FUNCTION "GLUE_SCALE" : VOID
TITLE =Glue Scale: DP Read, ASCII Parse, Valve Control, Alarms
// v0.11 - Simplified "Parse integer part" network: replaced the 7
//   duplicated digit-check blocks (Byte_0..Byte_6, one hand-unrolled
//   per byte, ~140 lines) with a single indirect-addressed loop over
//   Byte_0..Byte_5 plus a short unconditional block for Byte_6 - same
//   LAR1/+AR1/DBB[AR1,P#x.y] indirect-addressing idiom this project
//   already uses in FB1111/FB1112/FC130. Behavior is unchanged: leading
//   spaces are skipped until the first digit (FoundDigit latches once
//   set, matching v0.10), and Byte_6 - the field's last position - is
//   still always parsed unconditionally, space or not. Also dropped a
//   dead SET;=FoundDigit pair at the top that was immediately
//   overwritten by the following CLR;=FoundDigit two lines later.
//
// v0.12 changes vs v0.11 - synced against DB105 v0.3 (see that block's
//   changelog, and DB105_Online_1.xps captured 2026-09-17):
//   - NEW network "Detect scale fault": the KWS CY300 sends a fixed
//     sentinel value (all 7 digits of the Byte_0-6 field filled, no
//     leading spaces - confirmed live at 5222222) instead of a real
//     reading when its measurement goes negative. GrossWeight_Actual is
//     compared against DB105's new NegativeUnderScore_Value constant
//     every scan; a match latches Alarm_ScaleFault. Exact REAL equality
//     is safe here specifically because both sides are integer-valued
//     (no fractional digit) and well under 2^24 - bit-exact in IEEE754
//     single precision, not the usual float-equality trap.
//   - "Skip valve/alarm update" network now also gates on Alarm_ScaleFault,
//     same as ParseError - a scale reporting its fault sentinel is not
//     a real weight, so the valve must not react to it (freezes at
//     last-good state, same as a garbled telegram) until an operator
//     acknowledges/resets Alarm_ScaleFault via HMI (not yet wired - see
//     README "Still open", same gap as the two existing alarms).
//   - Valve control network retargeted from the retired Setpoint_Fill/
//     Hysteresis pair to DB105's new Fill_Start_SP/Fill_Stop_SP: opens
//     below Fill_Start_SP, closes at/above Fill_Stop_SP directly - no
//     Hysteresis subtraction needed since the two setpoints already
//     define the deadband.
//
// v0.13 changes vs v0.12 - HMI alarm reset (per DB105 v0.4):
//   - NEW network "Reset latched alarms", placed after the SKIP: label
//     so it always runs every scan regardless of this scan's
//     ParseError/Alarm_ScaleFault skip state - a latched alarm must
//     stay resettable even while it's actively freezing the rest of
//     this block, otherwise Alarm_ScaleFault could never be cleared
//     once it fires (it would perpetually skip past its own reset).
//     Reads DB105.Reset_Alarms directly (level, not edge) - clears
//     Alarm_Overfill/Alarm_Underfill/Alarm_ScaleFault together while
//     TRUE; each alarm's own network re-latches next scan if its fault
//     condition is still actually present, so this can't mask a live
//     fault by holding the button down.
VERSION : 0.13

VAR_TEMP
   RetVal1 : INT;
   RetVal2 : INT;
   IntPart : DINT;
   DecDigit : DINT;
   CharVal : INT;
   FoundDigit : BOOL;
   LoopIndex : INT;
END_VAR

BEGIN
NETWORK
TITLE =Read 16-byte consistent block (IB272-287) via DPRD_DAT

      CALL SFC  14 (
           LADDR                    := W#16#110,
           RET_VAL                  := #RetVal1,
           RECORD                   := P#DB4.DBX0.0 BYTE 16);

NETWORK
TITLE =Read 4-byte consistent block (IB289-292) via DPRD_DAT

      CALL SFC  14 (
           LADDR                    := W#16#121,
           RET_VAL                  := #RetVal2,
           RECORD                   := P#DB4.DBX16.0 BYTE 4);

NETWORK
TITLE =Validate telegram - check RetVal and fixed markers (decimal point, k, g)

      L     #RetVal1;
      L     0;
      <>I ;
      L     #RetVal2;
      L     0;
      <>I ;
      OW  ;
      L     "ABC3000A_DB".Byte_7;
      L     B#16#2E;
      <>I ;
      OW  ;
      L     "ABC3000A_DB".Byte_9;
      L     B#16#6B;
      <>I ;
      OW  ;
      L     "ABC3000A_DB".Byte_10;
      L     B#16#67;
      <>I ;
      OW  ;
      =     "GLUE_SCALE_CONTROL_DB".ParseError;

NETWORK
TITLE =Parse integer part, Byte_0-5 - loop, skip leading spaces until first digit

      CLR ;
      =     #FoundDigit;
      L     0;
      T     #IntPart;

      OPN   "ABC3000A_DB";
      LAR1  P#0.0;

      L     6;
LP1:  T     #LoopIndex;

      L     DBB [AR1,P#0.0];
      L     B#16#20;
      <>I ;
      S     #FoundDigit;

      A     #FoundDigit;
      JCN   ND1;

      L     DBB [AR1,P#0.0];
      L     B#16#30;
      -I  ;
      T     CharVal;
      L     #IntPart;
      L     10;
      *D  ;
      L     CharVal;
      ITD ;
      +D  ;
      T     #IntPart;

ND1:  +AR1  P#1.0;

      L     #LoopIndex;
      LOOP  LP1;

NETWORK
TITLE =Parse integer part, Byte_6 - field's last position, always a digit, no space check

      L     "ABC3000A_DB".Byte_6;
      L     B#16#30;
      -I  ;
      T     CharVal;
      L     #IntPart;
      L     10;
      *D  ;
      L     CharVal;
      ITD ;
      +D  ;
      T     #IntPart;

NETWORK
TITLE =Parse decimal digit (Byte_8) and build final REAL weight

      L     "ABC3000A_DB".Byte_8;
      L     B#16#30;
      -I  ;
      T     CharVal;
      L     CharVal;
      ITD ;
      T     #DecDigit;

      L     #IntPart;
      DTR ;
      T     "GLUE_SCALE_CONTROL_DB".GrossWeight_Actual;

      L     #DecDigit;
      DTR ;
      L     1.000000e+001;
      /R  ;
      L     "GLUE_SCALE_CONTROL_DB".GrossWeight_Actual;
      +R  ;
      T     "GLUE_SCALE_CONTROL_DB".GrossWeight_Actual;

NETWORK
TITLE =Detect scale fault - GrossWeight_Actual matches the scale's negative-value sentinel (latching)
// Exact REAL equality is safe here: both sides are integer-valued (no
// fractional digit) and well under 2^24, so the DTR conversion is
// bit-exact in IEEE754 single precision - this is not the usual
// float-equality trap.
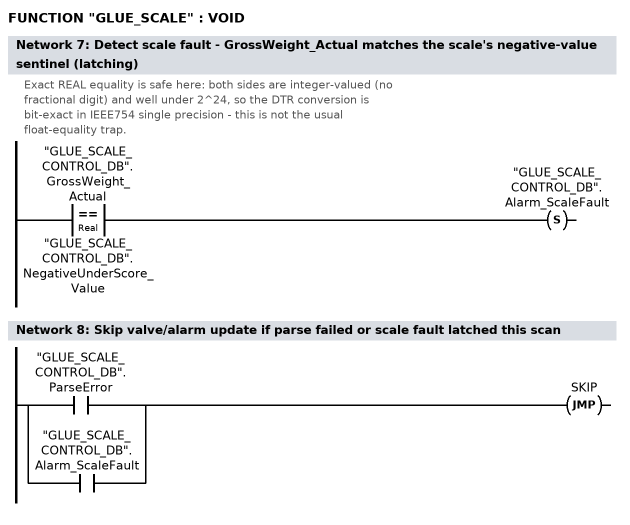
      L     "GLUE_SCALE_CONTROL_DB".GrossWeight_Actual;
      L     "GLUE_SCALE_CONTROL_DB".NegativeUnderScore_Value;
      ==R ;
      S     "GLUE_SCALE_CONTROL_DB".Alarm_ScaleFault;

NETWORK
TITLE =Skip valve/alarm update if parse failed or scale fault latched this scan

      A     "GLUE_SCALE_CONTROL_DB".ParseError;
      O     "GLUE_SCALE_CONTROL_DB".Alarm_ScaleFault;
      JC    SKIP;

NETWORK
TITLE =Valve control - open below Fill_Start_SP, close at/above Fill_Stop_SP

      A     "GLUE_SCALE_CONTROL_DB".Valve_Open;
      JC    CHKC;

      L     "GLUE_SCALE_CONTROL_DB".GrossWeight_Actual;
      L     "GLUE_SCALE_CONTROL_DB".Fill_Start_SP;
      <R  ;
      JC    OPEN;
      JU    VEND;

CHKC: L     "GLUE_SCALE_CONTROL_DB".GrossWeight_Actual;
      L     "GLUE_SCALE_CONTROL_DB".Fill_Stop_SP;
      >=R ;
      JC    CLOS;
      JU    VEND;

OPEN: SET ;
      S     "GLUE_SCALE_CONTROL_DB".Valve_Open;
      JU    VEND;

CLOS: SET ;
      R     "GLUE_SCALE_CONTROL_DB".Valve_Open;

VEND: NOP   0;

NETWORK
TITLE =Overfill alarm - latching, set on exceed, no auto-reset here
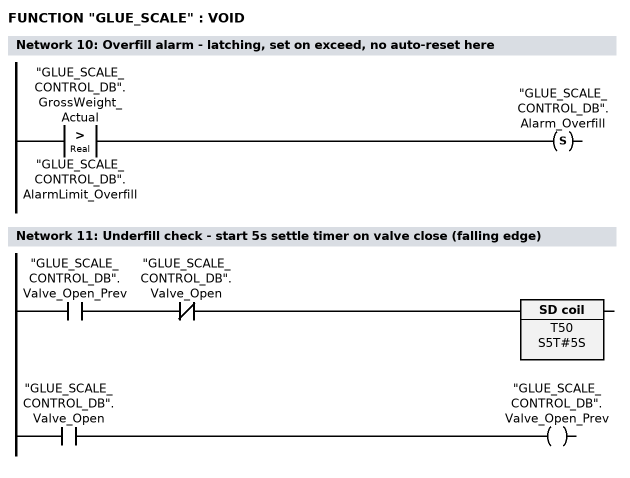

      L     "GLUE_SCALE_CONTROL_DB".GrossWeight_Actual;
      L     "GLUE_SCALE_CONTROL_DB".AlarmLimit_Overfill;
      >R  ;
      S     "GLUE_SCALE_CONTROL_DB".Alarm_Overfill;

NETWORK
TITLE =Underfill check - start 5s settle timer on valve close (falling edge)

      A     "GLUE_SCALE_CONTROL_DB".Valve_Open_Prev;
      AN    "GLUE_SCALE_CONTROL_DB".Valve_Open;
      L     S5T#5S;
      SD    T50;

      A     "GLUE_SCALE_CONTROL_DB".Valve_Open;
      =     "GLUE_SCALE_CONTROL_DB".Valve_Open_Prev;

NETWORK
TITLE =Underfill alarm - latch if weight still below limit when timer elapses

      A     T50;
      JCN   SKPU;
      L     "GLUE_SCALE_CONTROL_DB".GrossWeight_Actual;
      L     "GLUE_SCALE_CONTROL_DB".AlarmLimit_Underfill;
      <R  ;
      S     "GLUE_SCALE_CONTROL_DB".Alarm_Underfill;
SKPU: NOP   0;

NETWORK
TITLE =Exit point for parse-error skip

SKIP: NOP   0;

NETWORK
TITLE =Reset latched alarms - HMI-driven, runs regardless of this scan's skip state

      A     "GLUE_SCALE_CONTROL_DB".Reset_Alarms;
      R     "GLUE_SCALE_CONTROL_DB".Alarm_Overfill;
      R     "GLUE_SCALE_CONTROL_DB".Alarm_Underfill;
      R     "GLUE_SCALE_CONTROL_DB".Alarm_ScaleFault;

END_FUNCTION
